{attribute 'GeneratedUsingTerminal: EL3773-0000-0016'}
{attribute addProperty BoxType "EL3773-0000-0016"}
{attribute addProperty Id "AdsAddrAT %I*.TcoAmsAddr0DcOutputShiftAT %I*DINT4DcInputShiftAT %I*DINT4StateAT %I*UINT2"}
{attribute addProperty CRC "277399301"}
{attribute addProperty Size "10"}
TYPE InfoData_1088C705 :
STRUCT
	{attribute addProperty Name "AdsAddr"}
	AdsAddr AT %I* : .TcoAmsAddr;
	{attribute addProperty Name "DcOutputShift"}
	DcOutputShift AT %I* : DINT;
	{attribute addProperty Name "DcInputShift"}
	DcInputShift AT %I* : DINT;
	{attribute addProperty Name "State"}
	State AT %I* : UINT;
END_STRUCT
END_TYPE

(* stored: Version 1.2.0.0, ProductVersion 3.1.4024.9
   DUT InfoData_1088C705: Id {7e9b42da-8783-4dd3-abc0-ca0abf50f091} *)
